FUNCTION F_DimmAlgoForSwitch : INT
VAR_INPUT
	i_DimmingValue	: INT;
END_VAR
VAR_OUTPUT
	bTurnOffTheLight : BOOL := FALSE;
END_VAR
VAR
END_VAR

(*---------------------------------------------------------
Defines the Dimming Algorithm for dimmable Lights by standard switch
---------------------------------------------------------*)
IF i_DimmingValue > 192 THEN 	//Wenn Leuchtkraft > 75%
		i_DimmingValue := 192;
	ELSIF i_DimmingValue > 128 THEN //Wenn Leuchtkraft > 50%
		i_DimmingValue := 128;
	ELSIF i_DimmingValue > 64 THEN 	//Wenn Leuchtkraft > 25%
		i_DimmingValue := 64;
	ELSIF i_DimmingValue <= 64 THEN 	//Wenn Leuchtkraft bei 25%
		bTurnOffTheLight := TRUE;
	END_IF

F_DimmAlgoForSwitch := i_DimmingValue;

END_FUNCTION

(* stored: Version 1.1.0.1, ProductVersion 3.1.4024.4
   POU F_DimmAlgoForSwitch: Id {de034a1d-4341-4cd9-8548-0858c4708ecf}, SpecialFunc None *)
